{attribute 'linkalways'} 
{attribute 'no_explicit_call' := 'This FB is a CLASS and must be accessed using methods or properties'}
{attribute 'enable_dynamic_creation'}
FUNCTION_BLOCK FINAL EQ_LWORD EXTENDS Node
VAR
	in1 : _LWORD(0);
	in2 : _LWORD(0);
	out : _BOOL(FALSE);
END_VAR

METHOD PUBLIC Clone : I_Node
VAR
	pNode : POINTER TO EQ_LWORD;
END_VAR
pNode := __NEW(EQ_LWORD);
Clone := pNode^;
END_METHOD

METHOD FB_init : BOOL
VAR_INPUT
	bInitRetains : BOOL; // if TRUE, the retain variables are initialized (warm start / cold start)
	bInCopyCode : BOOL;  // if TRUE, the instance afterwards gets moved into the copy code (online change)
END_VAR
AddInput('in1',THIS^.in1);
AddInput('in2',THIS^.in2);
AddOutput('out', THIS^.out);
END_METHOD

METHOD PROTECTED OnExecute
VAR
END_VAR
out.Value := in1.Value = in2.Value;
END_METHOD

END_FUNCTION_BLOCK

(* stored: Version 1.1.0.1, ProductVersion 3.1.4024.15
   POU EQ_LWORD: Id {3eafbd5b-4617-4551-9f0f-52b07ca06454}, SpecialFunc None
   Folder Constructor: Id {bbce9c7e-e122-4051-8638-250872ca0163}
   Method Clone: Id {564c6ee0-cabb-4a2d-b2aa-13483b1dffba}
   Method FB_init: Id {0a39c18e-1398-49c7-b06f-fcbb73386e00}
   Method OnExecute: Id {d7157369-c7f1-4a82-a14e-243ab43a39bf} *)
